// TIA Portal V20 export
DATA_BLOCK "Cam_1"   // DB3, Motion_DB
// stored: InstanceOfName TO_Cam, OfSystemLibElement TO_Cam, OfSystemLibVersion 6.0
TO_Cam   // technology object, version 6.0
   // // inherited from TO_CamBase
   // // inherited from TO_Object
   // VAR
   //    InterpolationSettings { S7_SetPoint := 'True'} : TO_Cam_Struct_InterpolationSettings;
   //    StatusCam { ExternalWritable := 'False'; S7_SetPoint := 'True'} : TO_Cam_Struct_StatusCam;
   //    Point { S7_SetPoint := 'True'} : Array[1..1000] of TO_Cam_Struct_PointData;
   //    ValidPoint : Array[1..1000] of Bool;
   //    Segment { S7_SetPoint := 'True'} : Array[1..50] of TO_Cam_Struct_SegmentData;
   //    ValidSegment : Array[1..50] of Bool;
   //    StatusWord { ExternalWritable := 'False'} : DWord;
   //    ErrorWord { ExternalWritable := 'False'} : DWord;
   //    ErrorDetail { ExternalWritable := 'False'; S7_SetPoint := 'True'} : TO_Struct_ErrorDetail;
   //    WarningWord { ExternalWritable := 'False'} : DWord;
   // END_VAR
BEGIN
   InterpolationSettings.InterpolationMode := 1;
   Segment[2].xmin := 180.0;
   Segment[1].xmax := 180.0;
   Segment[2].xmax := 360.0;
   Segment[2].a0 := 350.0;
   Segment[1].a1 := -5.35891813843383E-15;
   Segment[2].a1 := 1.78630604614461E-14;
   Segment[1].a2 := 3.07021351681105E-16;
   Segment[2].a2 := -2.79110319710095E-17;
   Segment[1].a3 := 0.000600137174211246;
   Segment[2].a3 := -0.000600137174211251;
   Segment[1].a4 := -5.00114311842707E-06;
   Segment[2].a4 := 5.00114311842709E-06;
   Segment[1].a5 := 1.11136513742824E-08;
   Segment[2].a5 := -1.11136513742824E-08;
   ValidSegment[1..2] := true;
END_DATA_BLOCK
